# EPICS substitutions: sdgEliteApp/Db/sdgElite.substitutions
file sdgEliteCommon.template
{{None}}

file sdgEliteChan.template
{
pattern{ N, S }
       { 1, A }
       { 2, B }
       { 3, C }
       { 4, D }
       { 5, E }
       { 6, F }
       { 7, G }
       { 8, H }
}
